FUNCTION_BLOCK CM_DIN
VAR_INPUT
	PI_autoHigh : BOOL;
END_VAR
VAR_OUTPUT
END_VAR
VAR_IN_OUT
	Control_data : CM_DIN_UDT;
END_VAR

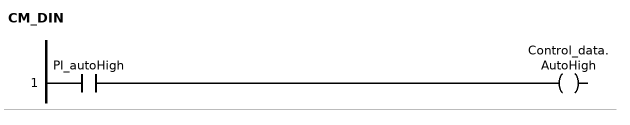
// NETWORK 1
Control_data.AutoHigh := PI_autoHigh;

END_FUNCTION_BLOCK

(* stored: Version 1.1.0.1, ProductVersion 3.1.4024.13
   POU CM_DIN: Id {e8489503-d724-46af-988b-da244bece43f}, SpecialFunc None *)
